Xinje XCPPro project, PLC1: XC5-32-4PLS (software 3.3j)

PROGRAM Ladder

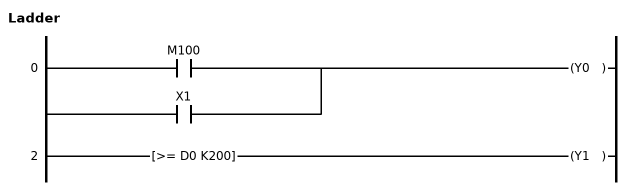
LD     M100
OR     X1
OUT    Y0
LD>=   D0 K200
OUT    Y1